TYPE ST_SafetyIO :
STRUCT
	Ch : ARRAY[1..4] OF BOOL  ; 
END_STRUCT
END_TYPE

(* stored: Version 1.1.0.1, ProductVersion 3.1.4024.12
   DUT ST_SafetyIO: Id {953519f6-8a39-4aaf-9a30-b2c98136ba0e} *)
